// TIA Portal V20 export
TYPE "LAxisCtrl_typeMoveVelocity"
TITLE = LAxisCtrl_typeMoveVelocity
// Support: tech.team.motioncontrol@siemens.com 
// Fax: +49 (0) 9131/98-1297
   STRUCT
      velocity : LReal := 0.0;   // Velocity/Speed for motion process (Value = 0.0: Permitted)
      acceleration : LReal := -1.0;   // Acceleration setpoint for motion process (Value > 0.0: The specified value is used; Value = 0.0: Not permitted; Value < 0.0: Use of the default value configured in the technology object)
      deceleration : LReal := -1.0;   // Deceleration setpoint for motion process (Value > 0.0: The specified value is used; Value = 0.0: Not permitted; Value < 0.0: Use of the default value configured in the technology object)
      jerk : LReal := -1.0;   // Jerk for velocity specification (Value > 0.0: Smooth velocity profile, the specified value is used; (Value = 0.0: Trapezoid velocity profile; (Value < 0.0: Use of the default value configured in the technology object)
      direction : Int := 0;   // Motion direction of the axis (0: The sign of the velocity parameter defines the direction; 1: Positive direction; 2: Negative direction)
      positionControlled : Bool := TRUE;   // TRUE: Position-controlled operation; FALSE: Non position-controlled operation
      velocityChangeOnTheFly : Bool := FALSE;   // TRUE: Changing velocity on-the-fly; FALSE: Velocity change requires a new rising edge on moveVelocity input
   END_STRUCT;
END_TYPE
